{attribute 'no-analysis'}
FUNCTION_BLOCK PLCopenNullRemote IMPLEMENTS IPLCopenCallRemote


// Copyright (c) 2024 Loupe (https://loupe.team), provided under the MIT License.


PROPERTY RemoteStatus : PLCopenStatusBase
GET
END_GET
SET
END_SET
END_PROPERTY


METHOD ReportAborted : BOOL

// Copyright (c) 2024 Loupe (https://loupe.team), provided under the MIT License.
END_METHOD

{attribute 'no-analysis'}
METHOD ReportErrored : BOOL
VAR_INPUT
  ID : INT;
END_VAR

// Copyright (c) 2024 Loupe (https://loupe.team), provided under the MIT License.
END_METHOD


METHOD ReportFinished : BOOL

// Copyright (c) 2024 Loupe (https://loupe.team), provided under the MIT License.
END_METHOD

END_FUNCTION_BLOCK

(* stored: Version 1.1.0.1
   POU PLCopenNullRemote: Id {73061230-7a8e-410b-ae26-c14eb801f0aa}, SpecialFunc None
   Property RemoteStatus: Id {84bb0023-487f-4833-ab3a-6bf154688ca2}
   Get Get: Id {3030317c-e694-4f80-994c-f5a95fac3c12}
   Set Set: Id {072515d1-b207-49fe-b993-f97b9c3f49cf}
   Method ReportAborted: Id {d3377050-9f4c-49f6-a051-4bcdc44d847d}
   Method ReportErrored: Id {97c3ac24-72bd-4b21-93c4-11f805822d38}
   Method ReportFinished: Id {6fdf66c9-5086-43d9-b213-c69b23218cc4} *)
